Staubli VAL3: Joint2Joint.pgx

public program Joint2Joint(jointRx x_jJSource, jointRx& x_jDest, bool& x_bRes)
  local pointRx l_p
begin

  //2015.09.08
  //更换这个运算
 // if TxtFile:fPofffset.trsf=={0,0,0,0,0,0} and TxtFile:fToffset.trsf=={0,0,0,0,0,0} and (TxtFile:fArray.trsf=={0,0,0,0,0,0} or TxtFile:fArray.trsf=={1,0,1,0,0,0})
 if TxtFile:fPofffset.trsf=={0,0,0,0,0,0} and TxtFile:fToffset.trsf=={0,0,0,0,0,0} and (TxtFile:fArray.trsf.x<2 and TxtFile:fArray.trsf.z<2)
    x_bRes=true
    x_jDest=x_jJSource

  else

    //Joint点的建立与frame无关，
    //joint点会偏移，当有Array
    l_p=jointToPoint(TxtFile:tCfg,world,x_jJSource)
    l_p.trsf=!TxtFile:fTraj.trsf*!TxtFile:fProduct.trsf*l_p.trsf
    link(l_p,TxtFile:fArray)

    x_bRes=pointToJoint(TxtFile:tCfg,x_jJSource,l_p,x_jDest)

  endIf








end
